// TIA Portal V17 export
// export: Created 2026-04-13T11:12:04.4957836Z, ExportSetting WithDefaults, DisplayName Totally Integrated Automation Portal, DisplayVersion V17 Update 4, DisplayName TIA Portal Openness, DisplayVersion V17 Update 4, DisplayName TIA Portal Version Control Interface, DisplayVersion V17, DisplayName SINAMICS Startdrive Advanced, DisplayVersion V17, DisplayName SINAMICS Startdrive G130, G150, S120, S150, SINAMICS MV, S210, DisplayVersion V17, DisplayName SINAMICS Startdrive G110M, G120, G120C, G120D, G120P, G115D, DisplayVersion V17, DisplayName STEP 7 Professional, DisplayVersion V17 Update 4, DisplayName STEP 7 Safety, DisplayVersion V17, DisplayName WinCC Professional, DisplayVersion V17 Update 4
FUNCTION_BLOCK "B4-清洗连锁"   // FB58, SCL
{ S7_Optimized_Access := 'TRUE' }
VERSION : 0.1
// stored: AutoNumber true, IsIECCheckEnabled false, IsRetainMemResEnabled false, MemoryReserve 100, SetENOAutomatically false, UDAEnableTagReadback false
   VAR
      TON0 : TON_TIME;
      TON1 : TON_TIME;
      TON2 { S7_SetPoint := 'True'} : TON_TIME;
      TON3 { S7_SetPoint := 'True'} : TON_TIME;
      TON4 { S7_SetPoint := 'True'} : TON_TIME;
      TON5 { S7_SetPoint := 'True'} : TON_TIME;
      TON6 { S7_SetPoint := 'True'} : TON_TIME;
      TON7 { S7_SetPoint := 'True'} : TON_TIME;
      R_TRIG { S7_SetPoint := 'True'} : Array[0..100] of R_TRIG;
      RT { S7_SetPoint := 'True'} : Array[0..100] of Bool;
      F_TRIG { S7_SetPoint := 'True'} : Array[0..100] of F_TRIG;
      FT { S7_SetPoint := 'True'} : Array[0..100] of Bool;
      BJ报警上升辅助 : Bool;
      BJ报警下降辅助 : Bool;
      BJ报警上升沿 { S7_SetPoint := 'True'} : R_TRIG;
      BJ报警下降沿 { S7_SetPoint := 'True'} : F_TRIG;
      F1 { S7_SetPoint := 'True'} : Bool;
      F2 : Bool;
      ET0 : Time;
      ET1 : Time;
      ET2 : Time;
      ET3 : Time;
      ET4 : Time;
      ET5 : Time;
      ET6 : Time;
      ET7 : Time;
      F3 : Bool;
      F4 : Bool;
      Temp_1 : Int;
      AERROR : Bool;
      t0_1s : TON_TIME;
      YC1 { S7_SetPoint := 'True'} : DInt;
      YC2 : DInt;
      YC3 : DInt;
      YC4 : DInt;
      YC5 : DInt;
   END_VAR
BEGIN
   IF "PW".MS模式设定 = 5.0 OR "PW".MS模式设定 = 6.0 OR "PW".MS模式设定 = 2.0 THEN

       IF "MFZ仿真调试" THEN
           IF "QQG气缸升" = 0 AND "QQG气缸降" = 1 THEN
               "IQX清洗伸缩气缸降反馈" := 1;
           END_IF;

           IF "QQG气缸升" = 1 AND "QQG气缸降" = 0 THEN
               "IQX清洗伸缩气缸升反馈" := 1;
           END_IF;

          (* IF "MQG气缸升" THEN
               "QQG气缸升" := 1;
           ELSE
               "QQG气缸升" := 0;
           END_IF;

           IF "MQG气缸降" THEN
               "QQG气缸降" := 1;
           ELSE
               "QQG气缸降" := 0;
           END_IF; *)

       END_IF;




       IF "ATD塔顶清洗球阀开报警" OR "ATD塔顶清洗球阀关报警" THEN
           #AERROR := 1;
       ELSE
           #AERROR := 0;
       END_IF;

       IF "MZT主塔伸缩气缸" THEN
           "MQG气缸升" := 0;
           "QQG气缸升" := 0;
           "MQG气缸降" := 1;
           "QQG气缸降" := 1;
       ELSE
           "MQG气缸升" := 1;
           "QQG气缸升" := 1;
           "MQG气缸降" := 0;
           "QQG气缸降" := 0;

       END_IF;


      (* #TON1(IN := "MTD塔顶清洗阀" AND NOT #AERROR,
             PT := T#5s,
             ET => #ET1);

       #TON2(IN := "MZT主塔伸缩气缸" AND #"QQ气缸下限位" AND NOT #AERROR AND "MTD塔顶清洗阀",
             PT := T#5s,
             ET => #ET2); *)

       IF "MZT主塔清洗"  THEN
           #YC3 := 0;
           #YC4 := 0;

           "MTD塔顶清洗球阀" := 1;
           "QTD塔顶清洗球阀" := 1;

           IF "QTD塔顶清洗球阀" AND #t0_1s.Q AND #YC1 < 10 THEN
               #YC1 := #YC1 + 1;
           END_IF;

           IF #YC1 >= 10.0 THEN
               "MZT主塔伸缩气缸" := 1;
               #YC1 := 0;
           END_IF;

           IF "IQX清洗伸缩气缸降反馈" AND #t0_1s.Q AND #YC2 < 10 THEN
               #YC2 := #YC2 + 1;
           END_IF;

           IF #YC2 >= 10 AND "MZT主塔清洗进水阀" THEN
               "MZT主塔清洗进水阀" := 1;
               "QZT主塔清洗进水阀" := 1;
               //"MTD塔顶清洗阀" := 1;
              // "QTD塔顶清洗阀" := 1;
           END_IF;
       END_IF;


       IF NOT "MZT主塔清洗" THEN
           #YC1 := 0;
           #YC2 := 0;
          // "MTD塔顶清洗阀" := 0;
          // "QTD塔顶清洗阀" := 0;
           "MZT主塔清洗进水阀" := 0;
           "QZT主塔清洗进水阀" := 0;

           IF NOT "QZT主塔清洗进水阀"  AND #t0_1s.Q AND #YC3 < 10 THEN
               #YC3 := #YC3 + 1;
           END_IF;

           IF #YC3 >= 10.0 AND NOT "QZT主塔清洗进水阀"  THEN
               "MZT主塔伸缩气缸" := 0;

           END_IF;

           IF "IQX清洗伸缩气缸升反馈" AND #t0_1s.Q AND #YC4 < 10 THEN
               #YC4 := #YC4 + 1;
           END_IF;

           IF #YC4 >= 10 AND "IQX清洗伸缩气缸升反馈" THEN
               "MTD塔顶清洗球阀" := 0;
               "QTD塔顶清洗球阀" := 0;
               #YC3 := 0;
               #YC4 := 0;
           END_IF;

       END_IF;

   END_IF;

   #t0_1s(IN := NOT #t0_1s.Q,
          PT := t#1000ms);
END_FUNCTION_BLOCK
